// TIA Portal V20 export
TYPE "type_emRelations_em4_cmStatus"
// stored: Access Published, Namespace Unit1
   STRUCT
      cmPnp1stAnodeDetect { S7_SetPoint := 'True'} : "LBC_typeDigitalSignalControlNode";
      cmPnp2ndAnodeDetect { ExternalAccessible := 'False'; ExternalVisible := 'False'; ExternalWritable := 'False'} : "LBC_typeDigitalSignalControlNode";
      cmAnodeAlignTableElectrodeDetect { ExternalWritable := 'False'} : "LBC_typeDigitalSignalControlNode";
      cmAnodeNgPnpElectrodeDetect { ExternalAccessible := 'False'; ExternalVisible := 'False'; ExternalWritable := 'False'; S7_SetPoint := 'True'} : "LBC_typeDigitalSignalControlNode";
      cmAnodeNgBoxFullSensorDetect { ExternalAccessible := 'False'; ExternalVisible := 'False'; ExternalWritable := 'False'; S7_SetPoint := 'True'} : "LBC_typeDigitalSignalControlNode";
      cmAnodeNgBoxDetect { ExternalAccessible := 'False'; ExternalVisible := 'False'; ExternalWritable := 'False'} : "LBC_typeDigitalSignalControlNode";
      cmAnodeMainPnP1AxisX { S7_SetPoint := 'True'} : "LBC_typeAxis64PosControlNode";
      cmAnodeMainPnP2AxisX { S7_SetPoint := 'True'} : "LBC_typeAxis64PosControlNode";
      cmAnodeMainPnP1AxisY { S7_SetPoint := 'True'} : "LBC_typeAxis64PosControlNode";
      cmAnodeMainPnP1AxisZ { S7_SetPoint := 'True'} : "LBC_typeAxis64PosControlNode";
      cmAnodeMainPnP2AxisZ { S7_SetPoint := 'True'} : "LBC_typeAxis64PosControlNode";
      cmAnodeAlignTableAxisX { S7_SetPoint := 'True'} : "LBC_typeAxis64PosControlNode";
      cmAnodeAlignTableAxisY1 { S7_SetPoint := 'True'} : "LBC_typeAxis64PosControlNode";
      cmAnodeAlignTableAxisY2 { S7_SetPoint := 'True'} : "LBC_typeAxis64PosControlNode";
      cmAnodeMainPnP1RotaryCwCcw { S7_SetPoint := 'True'} : "LBC_typeTwoWayActuatorControlNode";
      cmAnodeMainPnP1SuctionPlateVacuum { S7_SetPoint := 'True'} : "LBC_typeTwoWayActuatorControlNode";
      cmAnodeMainPnP2SuctionPlateVacuum { S7_SetPoint := 'True'} : "LBC_typeTwoWayActuatorControlNode";
      cmAnodeAlignTableSuctionPlateVacuum { S7_SetPoint := 'True'} : "LBC_typeTwoWayActuatorControlNode";
      cmAnodeGlassCleaning { S7_SetPoint := 'True'} : "LBC_typeTwoWayActuatorControlNode";
      cmAnodeNgPnpUpDown { S7_SetPoint := 'True'} : "LBC_typeTwoWayActuatorControlNode";
      cmAnodeNgPnp1stFwdBwd { S7_SetPoint := 'True'} : "LBC_typeTwoWayActuatorControlNode";
      cmAnodeNgPnp2ndFwdBwd { S7_SetPoint := 'True'} : "LBC_typeTwoWayActuatorControlNode";
      cmAnodeMaintenanceMovingFixFwdBwd { S7_SetPoint := 'True'} : "LBC_typeTwoWayActuatorControlNode";
      cmAnodeNgBoxLiftUpDown { S7_SetPoint := 'True'} : "LBC_typeTwoWayActuatorControlNode";
      cmAnodeNgBoxLockUpDown { S7_SetPoint := 'True'} : "LBC_typeTwoWayActuatorControlNode";
      cmAnodeNgPnpVaccum { S7_SetPoint := 'True'} : "LBC_typeTwoWayActuatorControlNode";
      cmAnodeConveyorCoverFwdBwd { S7_SetPoint := 'True'} : "LBC_typeTwoWayActuatorControlNode";
      cmAnodeConveyorPickUpBlower { S7_SetPoint := 'True'} : "LBC_typeTwoWayActuatorControlNode";
      cmAnodeVisionControllerInterface { S7_SetPoint := 'True'} : "LER_typeVisionControlNode";
   END_STRUCT;
   // cmPnp1stAnodeDetect.commands.reset := FALSE;
   // cmPnp1stAnodeDetect.commands.simulation := FALSE;
   // cmPnp1stAnodeDetect.commands.quality := TRUE;
END_TYPE
